{attribute 'qualified_only'}
VAR_GLOBAL	
	ASCII AT %I*: BYTE; 	// ASCII Code des Zeichens
END_VAR

(* stored: Version 1.1.0.1, ProductVersion 3.1.4024.4
   GVL SimDI: Id {c2d05302-d374-4f85-80dd-41006a3e3277} *)
